FUNCTION sMsg_Process_Buffer : BOOL
VAR_IN_OUT
    pBuffer   : ST_Msg_Buffer;
END_VAR
VAR
    ptr     :UDINT;
    len     :UDINT;
END_VAR

IF pBuffer.Ack THEN
    pBuffer.Ack := FALSE;
    pBuffer.Ready := FALSE;
    pBuffer.Sending[IDX0] := 0;    // effectively indicates the buffer is empty
    pBuffer.WatchDogTmr := 0;
	pBuffer.Stats.ACKcnt := pBuffer.Stats.ACKcnt + 1;
	IF (pBuffer.Stats.ACKcnt >= 2147483500) THEN
		pBuffer.Stats.ACKcnt := 1;
	END_IF
	
END_IF

// if there is something pending and the sending is empty...
IF pBuffer.Pending[IDX0] > 0 AND pBuffer.Sending[IDX0] = 0 THEN
    // ... transfer pending to sending
    ptr := 0;
    WHILE pBuffer.Pending[ptr] > 0 AND ptr < 4000 DO
        pBuffer.Sending[ptr] := pBuffer.Pending[ptr];
        pBuffer.Pending[ptr] := 0;      // erase as we go along
        ptr := ptr + 1;
	END_WHILE
    pBuffer.Sending[ptr] := 0;   // don't forget to zero terminate the string
    
	pBuffer.Stats.RDYcnt := pBuffer.Stats.RDYcnt + 1;
	IF (pBuffer.Stats.RDYcnt >= 2147483500) THEN
		pBuffer.Stats.RDYcnt := 1;
	END_IF
	pBuffer.Ready := TRUE;
    pBuffer.WatchDogTmr := 0;     // time how long it takes to pick up this msg
END_IF
//(* removing the watchdog per Mike Higleys request. He states that toggling the Ready bit messes with the services - mjm
// if the sending buffer is active with data... 
IF pBuffer.Sending[IDX0] > 0 THEN
    // time how long until it's picked up
    pBuffer.WatchDogTmr := pBuffer.WatchDogTmr + 1;
    // if not within the timeout...   (25 = 100ms)
    IF pBuffer.WatchDogTmr = 25 THEN
        // toggle the Ready bit OFF
        pBuffer.Ready := FALSE;
		pBuffer.Stats.WatchdofTimeoutCnt := pBuffer.Stats.WatchdofTimeoutCnt + 1;
	END_IF
    IF pBuffer.WatchDogTmr = 51 THEN
        pBuffer.Ready := TRUE;
        pBuffer.WatchDogTmr := 0;
	END_IF
END_IF
//*)

END_FUNCTION

(* stored: Version 1.1.0.1, ProductVersion 3.1.4024.9
   POU sMsg_Process_Buffer: Id {fdccdcbe-c5a8-4c31-92e6-7e0bd34d7c67}, SpecialFunc None *)
